// TwinCAT 3 PLC project PLC1
// ProgramVersion: 3.1.4026.18
// CompilerDefines: VISU_USEPROPERTYINFO
// libraries:
//   [LoggedEventsToPLC], * (Beckhoff Automation LLC.)
//   Tc2_Standard, * (Beckhoff Automation GmbH)
//   Tc2_System, * (Beckhoff Automation GmbH)
//   Tc2_Utilities, * (Beckhoff Automation GmbH)
//   Tc3_EventLogger, * (Beckhoff Automation GmbH)
//   VisuElemEventTable, * (System)
//   VisuSymbols, 4.5.0.0 (System)
// project tree:
//   / GlobalTextList.TcGTLO (not stored), PlcTask.TcTTO (not stored), Visualization Manager.TcVMO (not stored), VISU_TASK.TcTTO (not stored)
//   POUs/ MAIN.TcPOU, PRG_GenerateEvents.TcPOU
//   VISUs/ Visualization.TcVIS (not stored)

// ---- POUs/MAIN.TcPOU
PROGRAM MAIN
VAR
	// FB_ReadTc3Events
	fbReadTc3Events	   : FB_ReadTc3Events2;
	bReadEvents		   : BOOL							   := TRUE;
	nLanguage		   : DINT							   := 1033;
	eDateAndTimeFormat : Tc2_Utilities.E_DateAndTimeFormat := Tc2_Utilities.E_DateAndTimeFormat.en_US;
	bClearDisplay	   : BOOL;
	eSeverityMin	   : TcEventSeverity;
	bError			   : BOOL;
	hr				   : HRESULT;
	numOfEvents		   : UDINT;
	ReadLoggedEvents   : BOOL;
	Loaded			   : BOOL;
	Result			   : HRESULT;
END_VAR

// Call fbReadTc3Events
fbReadTc3Events(bReadEvents		   := bReadEvents,
				nLanguageID		   := nLanguage,
				eDateAndTimeFormat := eDateAndTimeFormat,
				bClearTable		   := bClearDisplay,
				bClearLoggedTable  := bClearDisplay,
				eMinSeverity	   := eSeverityMin,
				nNumberOfEvents	   => numOfEvents,
				bError			   => bError,
				hrErrorCode		   => hr);

bClearDisplay := FALSE;

IF ReadLoggedEvents THEN
	Loaded:=fbReadTc3Events.ReadLoggedEvents(bExec:=ReadLoggedEvents , hrErrorCode=>Result );
END_IF

END_PROGRAM

// ---- POUs/PRG_GenerateEvents.TcPOU
PROGRAM PRG_GenerateEvents
VAR
	Msg			  : ARRAY[1..5] OF FB_TcMessage;
	Alarm		  : ARRAY[1..5] OF FB_TcAlarm;
	i			  : INT;
	Init		  : BOOL := TRUE;
	RaiseAlarms	  : BOOL := FALSE;
	SendMsgs	  : BOOL := FALSE;
	ClearAlarms	  : BOOL := FALSE;
	ConfirmAlarms : BOOL := FALSE;
	Cnt			  : UDINT;

	//One alarm
	RaiseOneAlarm	: BOOL;
	ClearOneAlarm	: BOOL;
	ClearWithTrue	: BOOL;
	ConfirmOneAlarm : BOOL;
	Index			: INT := 1;
	SendOneMsg		: BOOL;
END_VAR

IF Init THEN
	Init := FALSE;

	//Messages
	Msg[1].CreateEx(stEventEntry := TC_EVENTS.MsgEvents.VerboseMsg);
	Msg[2].CreateEx(stEventEntry := TC_EVENTS.MsgEvents.InfoMsg);
	Msg[3].CreateEx(stEventEntry := TC_EVENTS.MsgEvents.WarningMsg);
	Msg[4].CreateEx(stEventEntry := TC_EVENTS.MsgEvents.ErrorMsg);
	Msg[5].CreateEx(stEventEntry := TC_EVENTS.MsgEvents.CriticalMsg);

	//Alarms
	Alarm[1].CreateEx(stEventEntry := TC_EVENTS.AlarmEvents.VerboseAlarm, bWithConfirmation := TRUE);
	Alarm[2].CreateEx(stEventEntry := TC_EVENTS.AlarmEvents.InfoAlarm, bWithConfirmation := TRUE);
	Alarm[3].CreateEx(stEventEntry := TC_EVENTS.AlarmEvents.WarningAlarm, bWithConfirmation := FALSE);
	Alarm[4].CreateEx(stEventEntry := TC_EVENTS.AlarmEvents.ErrorAlarm, bWithConfirmation := FALSE);
	Alarm[5].CreateEx(stEventEntry := TC_EVENTS.AlarmEvents.CriticalAlarm, bWithConfirmation := FALSE);
END_IF

IF RaiseAlarms THEN
	RaiseAlarms := FALSE;
	Cnt			:= Cnt + 1;
	FOR i := 1 TO 5 DO
		Alarm[i].ipArguments.Clear().AddUDInt(Cnt);
		Alarm[i].Raise();
	END_FOR
END_IF

IF SendMsgs THEN
	SendMsgs := FALSE;
	Cnt		 := Cnt + 1;
	FOR i := 1 TO 5 DO
		Msg[i].ipArguments.Clear().AddUDInt(Cnt);
		Msg[i].Send();
	END_FOR
END_IF

IF ConfirmAlarms THEN
	ConfirmAlarms := FALSE;
	FOR i := 1 TO 5 DO
		Alarm[i].Confirm();
	END_FOR
END_IF

IF ClearAlarms THEN
	ClearAlarms := FALSE;
	FOR i := 1 TO 5 DO
		Alarm[i].Clear();
	END_FOR
END_IF

IF RaiseOneAlarm THEN
	RaiseOneAlarm := FALSE;
	Alarm[Index].ipArguments.Clear().AddUDInt(Cnt);
	Alarm[Index].Raise();
END_IF

IF ClearOneAlarm THEN
	ClearOneAlarm := FALSE;
	Alarm[Index].Clear();
END_IF

IF ClearWithTrue THEN
	ClearWithTrue := FALSE;
	Alarm[Index].Clear(0, TRUE);
END_IF

IF ConfirmOneAlarm THEN
	ConfirmOneAlarm := FALSE;
	Alarm[Index].Confirm();
END_IF

IF SendOneMsg THEN
	SendOneMsg := FALSE;
	Msg[Index].ipArguments.Clear().AddUDInt(Cnt);
	Msg[Index].Send();
END_IF

END_PROGRAM
